// TIA Portal V20 export
TYPE "typeSequenceControlNodeJobInterface_sideTapeFixStage"
// stored: Namespace Unit1.Em4
   STRUCT
      loadJob2 : "LER_typeJobInterface";
      taping1Job3 : "LER_typeJobInterface";
      taping2Job4 : "LER_typeJobInterface";
      taping3Job5 : "LER_typeJobInterface";
      taping4Job6 : "LER_typeJobInterface";
      unloadJob7 : "LER_typeJobInterface";
   END_STRUCT;
END_TYPE
